ABB RAPID module: Wobj_wobj_A3.mod

MODULE Wobj_wobj_A3
	! Points are read in order of declaration.
  ! Please do not change the order of points!

  LOCAL PERS robtarget pWobj_U_PointX1:=[[1148.649,-1271.473,-658.1318],[0.000886961061041802,0.694058060646057,0.719859719276428,0.00919583532959223],[-1,0,0,0],[0,9E+09,9E+09,9E+09,9E+09,9E+09]];
	LOCAL PERS robtarget pWobj_U_PointX2:=[[1180.568,-2074.475,-653.9741],[0.00088916253298521,0.694056928157806,0.719860851764679,0.00919465161859989],[-1,0,0,0],[0,9E+09,9E+09,9E+09,9E+09,9E+09]];
	LOCAL PERS robtarget pWobj_U_PointY1:=[[1879.346,-2048.435,-651.1993],[0.000889677961822599,0.694057822227478,0.719859957695007,0.0091954730451107],[-1,0,0,0],[0,9E+09,9E+09,9E+09,9E+09,9E+09]];

ENDMODULE
